// SIMATIC STEP 7 (V5.x) project Lift
// CPU: CPU315-2 PN/DP(1)
// station: P_ADR_BUS
// station: Hardware
// station: SIMATIC 300 Station
// program: S7 Program(1)

SYMBOL_TABLE
"Номер этажа"	FB 1	FB 1	// Обработка номера этажа в зависимости от нажатия кнопок
"Позиционирование"	FC 1	FC 1	// Позицтонирование лифта в зависимости от задания
"Управление дверями"	FC 2	FC 2	// Открытие и закрытие дверей
"Закрыть двери"	FC 3	FC 3	// Закрыть все двери
"IN_4...20_MA"	FC 4	FC 4	// ANALOG INPUT 4...20 MA
"ReadyDoor"	M 0.0	BOOL	// Готовность дверей
"ReadyFloor"	M 0.1	BOOL	// Приехали на этаж, который нужно
"Program_1"	M 1.0	BOOL	// Программа 1
"Program_2"	M 1.1	BOOL	// Программа 2
"Speed"	MD 200	DWORD	// Скорость лифта
"NumberFloor"	MW 100	INT	// Номер этажа
"NumberFloor_1"	MW 102	INT	// Номер этажа 1
"NumberFloor_2"	MW 104	INT	// Номер этажа 2
"Главный цикл"	OB 1	OB 1
"Open_Door_1"	Q 1.0	BOOL	// Открыть двери 1
"Door_1_Close"	Q 1.1	BOOL	// Закрыть двери на первом этаже
"Open_Door_2"	Q 1.2	BOOL	// Открыть двери 2
"Door_2_Close"	Q 1.3	BOOL	// Закрыть двери на втором этаже
"Open_Door_3"	Q 1.4	BOOL	// Открыть двери 3
"Door_3_Close"	Q 1.5	BOOL	// Закрыть двери на третьем этаже
"Open_Door_4"	Q 1.6	BOOL	// Открыть двери кабины лифта
"Door_4_Close"	Q 1.7	BOOL	// Закрыть двери внутри лифта
"READ_SI"	SFC 105	SFC 105	// Reading Dynamically Assigned System Instances
END_SYMBOL_TABLE

FUNCTION_BLOCK "Номер этажа"	// FB 1
VERSION : 0.1
VAR_INPUT
  ReadyFloor : BOOL ;	//Мы находимся на том этаже, котором нужно
END_VAR
VAR_TEMP
  NumberFloor_1 : INT ;	//Переменная, хранящая номер этажа при нажатии кнопок внутри лифта
  NumberFloor_2 : INT ;	//Переменная, хранящая номер этажа при нажатии кнопок снаружи лифта
END_VAR
BEGIN
NETWORK
TITLE = Выбор этажа при нажатии кнопки внутри лифта
//Первый этаж
      A     I 0.0;
      JCN   M1;
      L     1;
      T     "NumberFloor_1";
      S     "Program_1";
M1:   NOP   0;
//Второй этаж
      A     I 0.1;
      JCN   M2;
      L     2;
      T     "NumberFloor_1";
      S     "Program_1";
M2:   NOP   0;
// Третий этаж
      A     I 0.2;
      JCN   M3;
      L     3;
      T     "NumberFloor_1";
      S     "Program_1";
M3:   NOP   0;
NETWORK
TITLE = Выбор этажа при нажатии кнопки со стороны подъезда
      A     I 0.4;
      JCN   M4;
      L     1;
      T     "NumberFloor_2";
      S     "Program_2";
M4:   NOP   0;
      O     I 0.5;
      O     I 0.6;
      JCN   M5;
      L     2;
      T     "NumberFloor_2";
      S     "Program_2";
M5:   NOP   0;
      A     I 0.7;
      JCN   M6;
      L     3;
      T     "NumberFloor_2";
      S     "Program_2";
M6:   NOP   0;
NETWORK
TITLE = Управление этажами
//Если работает программа 1, тогда передаем номер
//этажа с внутренних кнопок
      A     "Program_1";
      JCN   M7;
      L     "NumberFloor_1";
      T     "NumberFloor";
M7:   NOP   0;
//Если работает программа 2, тогда передаем номер
//этажа с внешних кнопок
      A     "Program_2";
      AN    "Program_1";
      JCN   M8;
      L     "NumberFloor_2";
      T     "NumberFloor";
M8:   NOP   0;
NETWORK
TITLE = Сброс Program_2
      A     I 1.6;
      FP    M 1.2;
      AN    "Program_1";
      A     "Program_2";
      R     "Program_2";
NETWORK
TITLE = Сброс Program_1
      A     I 1.6;
      FP    M 1.5;
      A     "Program_1";
      R     "Program_1";
END_FUNCTION_BLOCK

FUNCTION "Позиционирование" : VOID	// FC 1
TITLE = Устанока задания скорости лифта
VERSION : 0.1
VAR_INPUT
  NumberFloor : INT ;	//Установка номера этажа
  ReadyDoor : BOOL ;	//Готовность дверей для начала движения
END_VAR
VAR_OUTPUT
  Speed : DWORD ;	//Установка скорости для точного позиционировония
  ReadyFloor : BOOL ;	//Бит о том, что приехали на нужный этаж
END_VAR
VAR_TEMP
  SetPoint : DWORD ;	//Уставка высоты, на которую должен переместиться лифт
  ErrorValue : DWORD ;	//Величина ошибки
  PIW256_DWORD : DWORD ;	//Величина из входа преобразованная в двойное слово
  PIW256_REAL : REAL ;	//Величина из входа преобразованная в Real
END_VAR
BEGIN
NETWORK
TITLE = Установка задания высоты
//Устанока высоты первого жтажа
      L     #NumberFloor;
      L     1;
      ==I;
      JCN   M1;
      L     26994;
      T     #SetPoint;
M1:   NOP   0;
//Устанока высоты второго этажа
      L     #NumberFloor;
      L     2;
      ==I;
      JCN   M2;
      L     13500;
      T     #SetPoint;
M2:   NOP   0;
//Устанока высоты третьего этажа
      L     #NumberFloor;
      L     3;
      ==I;
      JCN   M3;
      L     4;
      T     #SetPoint;
M3:   NOP   0;
NETWORK
TITLE = Пеобразовать PIW 256 из WORD в DWORD 
      L     PIW 256;
      ITD;
      T     #PIW256_DWORD;
NETWORK
TITLE = Вычисление величины ошибки регулятора
      L     #PIW256_DWORD;
      L     #SetPoint;
      -D;
      T     #ErrorValue;
NETWORK
TITLE = Пропорциональная составляющая
//Задаем скорость на движение лифта в зависимости от ошибки регулятора. Если нет 
//разрешения на движение или номер этажа установлен в "0", тогда пропускаем этот 
//шаг
      O(;
      L     #NumberFloor;
      L     0;
      ==I;
      );
      ON    #ReadyDoor;
      JC    M4;
      L     #ErrorValue;
      T     #Speed;
M4:   NOP   0;
NETWORK
TITLE = Интегральная составляющая
//     L     #ErrorValue
//     L     #ErrorValue
//     +D    
NETWORK
TITLE =  Сброс временных переменных перед началом сравнения
//Сбрасываем временные вспомогательные переменные
      O     I 0.0;
      O     I 0.1;
      O     I 0.2;
      O     I 0.4;
      O     I 0.5;
      O     I 0.6;
      O     I 0.7;
      R     #ReadyFloor;
NETWORK
TITLE = Ограничение скорости движения лифта
      L     #Speed;
      L     L#2000;
      >D;
      JCN   M5;
      L     L#2000;
      T     #Speed;
M5:   NOP   0;
      L     #Speed;
      L     L#-2000;
      <D;
      JCN   M6;
      L     L#-2000;
      T     #Speed;
M6:   NOP   0;
NETWORK
TITLE = Обнуление задания скорости при отсутствии готовности дверей 
//Если нет разрешения на движение лифта или номер выбранного этажа равен 0, тогда 
//скорость равна нулю
      O(;
      L     #NumberFloor;
      L     0;
      ==I;
      );
      ON    #ReadyDoor;
      JCN   M7;
      L     0;
      T     #Speed;
M7:   NOP   0;
NETWORK
TITLE = Готовность этажа
//Если появился позитивный фронт выражения #ErrorValue == 0, тогда считает, 
//что мы приехали на нужный этаж
//Если задание соответствует актуальной позиции
      L     #PIW256_DWORD;
      L     #SetPoint;
      ==D;
      JCN   M8;
      S     #ReadyFloor;
M8:   NOP   0;
//Если задание не соответствует актуальной позиции
      L     #PIW256_DWORD;
      L     #SetPoint;
      ==D;
      JC    M9;
      R     #ReadyFloor;
M9:   NOP   0;
END_FUNCTION

FUNCTION "Управление дверями" : VOID	// FC 2
TITLE = Управление дверями
//Открывание и закрывание  дверей
VERSION : 0.1
VAR_INPUT
  ReadyFloor : BOOL ;	//ГПриехали на нужный этаж и можно открывать двери
  NumberFloor : INT ;	//Номер этажа
END_VAR
VAR_OUTPUT
  ReadyDoor : BOOL ;	//Готовность дверей для начала движения
END_VAR
VAR_TEMP
  NemberFloorNew : INT ;	//Новое значение этажа (для отслеживания изменения этажа)
  NemberFloorOld : INT ;	//Старое значение этажа (для отслеживания изменения этажа)
END_VAR
BEGIN
NETWORK
TITLE = Открывание дверей на первом этаже
//Если мы приехали на первый этаж, то открываем двери
      L     #NumberFloor;
      L     1;
      ==I;
      JCN   M1;
      A     #ReadyFloor;
      FP    M 0.2;
      S     "Open_Door_1";
      S     "Open_Door_4";
M1:   NOP   0;
NETWORK
TITLE = Открывание дверей на втором этаже
//Если мы приехали на второй этаж, то открываем двери
      L     #NumberFloor;
      L     2;
      ==I;
      JCN   M2;
      A     #ReadyFloor;
      FP    M 0.3;
      S     "Open_Door_2";
      S     "Open_Door_4";
M2:   NOP   0;
NETWORK
TITLE = Открывание дверей на третьем этаже
//Если мы приехали на тертий этаж, то открываем двери
      L     #NumberFloor;
      L     3;
      ==I;
      JCN   M3;
      A     #ReadyFloor;
      FP    M 0.4;
      S     "Open_Door_3";
      S     "Open_Door_4";
M3:   NOP   0;
NETWORK
TITLE = Закрытие дверей кабины лифта
//    O     "Door_3_Close"
//      O     "Door_2_Close"
//      O     "Door_1_Close"
//      FP    M      0.6
//     S     "Door_4_Close"
NETWORK
TITLE = Управление дверями от внешних кнопок (снаружи лифта)
//Если мы на первом этаже, нажали кнопку снаружи,
//тогда открываем двери лифта
      L     #NumberFloor;
      L     1;
      ==I;
      JCN   M4;
      A     I 0.4;
      A     #ReadyFloor;
      S     "Open_Door_1";
M4:   NOP   0;
//Если мы на втором этаже, нажали кнопку снаружи,
//тогда открываем двери лифта
      L     #NumberFloor;
      L     2;
      ==I;
      JCN   M5;
      A(;
      O     I 0.6;
      O     I 0.5;
      );
      A     #ReadyFloor;
      S     "Open_Door_2";
M5:   NOP   0;
//Если мы на третьем этаже, нажали кнопку снаружи,
//тогда открываем двери лифта
      L     #NumberFloor;
      L     3;
      ==I;
      JCN   M6;
      A     I 0.7;
      A     #ReadyFloor;
      S     "Open_Door_3";
M6:   NOP   0;
NETWORK
TITLE = Закрыть двери
      O     I 0.0;
      O     I 0.1;
      O     I 0.2;
      O     I 0.4;
      O     I 0.5;
      O     I 0.6;
      O     I 0.7;
      JCN   M7;
      CALL  "Закрыть двери";
M7:   NOP   0;
NETWORK
TITLE = Сброс задания на движение дверей лифта по концевикам 
//Если дверь достигла конечной нижней позиции, тогда сбрасываем задание на 
//закрывание или открывания этих дверей
      A     I 1.0;
      R     "Open_Door_1";
      A     I 1.1;
      R     "Door_1_Close";
      A     I 1.2;
      R     I 1.2;
      A     I 1.3;
      R     "Door_2_Close";
      A     I 1.4;
      R     "Open_Door_3";
      A     I 1.5;
      R     "Door_3_Close";
      A     I 1.6;
      R     "Open_Door_4";
      A     I 1.7;
      R     "Door_4_Close";
NETWORK
TITLE = Закрывание дверей после выполнения программы 1 или программы 2
      O     "Program_1";
      O     "Program_2";
      FN    M 1.3;
      L     S5T#3S;
      SF    T 0;
      A     T 0;
      FN    M 1.4;
      JCN   M8;
      CALL  "Закрыть двери";
M8:   NOP   0;
NETWORK
TITLE = Готовность дверей (разрешение на движение лифта)
//Если все двери закрыты, то передаем готовность дверей для разрешения на начало 
//движения
      A     I 1.1;
      A     I 1.3;
      A     I 1.5;
      A     I 1.7;
      =     #ReadyDoor;
END_FUNCTION

FUNCTION "Закрыть двери" : VOID	// FC 3
TITLE = Закрытие дверей
VERSION : 0.1
BEGIN
NETWORK
TITLE = Если нет концевика, то открываем двери
      R     "Open_Door_3";
      R     "Open_Door_2";
      R     "Open_Door_1";
      R     "Open_Door_4";
      AN    I 1.1;
      S     "Door_1_Close";
      AN    I 1.3;
      S     "Door_2_Close";
      AN    I 1.5;
      S     "Door_3_Close";
      AN    I 1.7;
      S     "Door_4_Close";
NETWORK
TITLE = Если наехали на концевик, тогда останавливаем открытие дверей
      A     I 1.1;
      R     "Door_1_Close";
      A     I 1.3;
      R     "Door_2_Close";
      A     I 1.5;
      R     "Door_3_Close";
      A     I 1.7;
      R     "Door_4_Close";
END_FUNCTION

DATA_BLOCK DB 1
VERSION : 0.0
"Номер этажа"
BEGIN
END_DATA_BLOCK

ORGANIZATION_BLOCK "Главный цикл"	// OB 1
TITLE = "Main Program Sweep (Cycle)"
VERSION : 0.1
VAR_TEMP
  OB1_EV_CLASS : BYTE ;	//Bits 0-3 = 1 (Coming event), Bits 4-7 = 1 (Event class 1)
  OB1_SCAN_1 : BYTE ;	//1 (Cold restart scan 1 of OB 1), 3 (Scan 2-n of OB 1)
  OB1_PRIORITY : BYTE ;	//Priority of OB Execution
  OB1_OB_NUMBR : BYTE ;	//1 (Organization block 1, OB1)
  OB1_RESERVED_1 : BYTE ;	//Reserved for system
  OB1_RESERVED_2 : BYTE ;	//Reserved for system
  OB1_PREV_CYCLE : INT ;	//Cycle time of previous OB1 scan (milliseconds)
  OB1_MIN_CYCLE : INT ;	//Minimum cycle time of OB1 (milliseconds)
  OB1_MAX_CYCLE : INT ;	//Maximum cycle time of OB1 (milliseconds)
  OB1_DATE_TIME : DATE_AND_TIME ;	//Date and time OB1 started
END_VAR
BEGIN
NETWORK
TITLE =
      L     "NumberFloor";
      L     0;
      ==I;
      JCN   M1;
      S     "Door_3_Close";
      S     "Door_2_Close";
      S     "Door_1_Close";
      S     "Door_4_Close";
M1:   NOP   0;
NETWORK
TITLE =
      CALL  "Номер этажа" , DB 1 (
           ReadyFloor               := "ReadyFloor");
      CALL  "Позиционирование" (
           NumberFloor              := "NumberFloor",
           ReadyDoor                := "ReadyDoor",
           Speed                    := "Speed",
           ReadyFloor               := "ReadyFloor");
      CALL  "Управление дверями" (
           ReadyFloor               := "ReadyFloor",
           NumberFloor              := "NumberFloor",
           ReadyDoor                := "ReadyDoor");
END_ORGANIZATION_BLOCK
